{attribute 'qualified_only'}
VAR_GLOBAL
	eEventTraceLevel : TcEventSeverity := TcEventSeverity.Critical;  
END_VAR

(* stored: Version 1.1.0.1, ProductVersion 3.1.4022.10
   GVL GVL: Id {2205f020-c552-4553-98ed-4e2509e55bed} *)
